Staubli VAL3: AlignPage.pgx

public program AlignPage(tool x_tTool)
  local num l_nKey
  local string l_sButton[2]
  local num l_i
  local bool l_bAlignDone
  local bool l_bExit
  local string l_sYesNo
begin
  //-----------------------------------------------------------------------
  //Header begin
  //Description of program
  //  工具对齐界面
  //  F1:终止
  //Input parameters
  //  tool x_tTool:工具值
  //Output paramaters
  //Example
  //  call Align(tool)
  //History
  //  Creation : 2012-06-11 - PF.Zhong
  //Header end
  //-----------------------------------------------------------------------
  cls()
  bAlignDone=false
  l_bExit=false
  taskCreate "Align",30,Align(x_tTool,bAlignDone)
  delay(0.1)
  while !bAlignDone and !l_bExit
      call user:timerDialog("机器人工具头正在对齐，请按住Move/Hold键",0)
      call user:typeLen(1,13,"终止",4)
      l_nKey=getKey()
      switch l_nKey
        case 271
          //终止
          cls()
          l_sButton[0]="是"
          l_sButton[1]="否"
          call user:questionDialog("是否终止对齐?",l_sButton,l_i)
          if l_i==0 or l_i==1
            resetMotion()
            stopMove()
            taskKill("Align")
            l_bExit=true
          else
            cls()
          endIf
        break
      endSwitch
      delay(0)
  endWhile
  if bAlignDone
    l_sYesNo="确定"
    call user:yes("对齐完毕!",l_sYesNo)
  else
    l_sYesNo="确定"
    call user:yes("对齐未完成!",l_sYesNo)
  endIf
end
